(* CoDeSys 2.3.9.55 project: BarCode.pro *)
(* Libraries: STANDARD.LIB 2.6.14 11:37:46, IECSFC.LIB 2.6.14 11:37:46, ANALYZATION.LIB 2.6.14 11:37:46 *)

(* PLC configuration (modules and I/O channels)
PLC63 [Root] node -1, in %IB0 out %QB0 {BName = #NМеню ПЛК63#A0; MinCycleLenght = 1; MaxCycleLenght = 1000}
  Configuration [ID10050] node 0, in %IB0 out %QB0 {BName = #NКонфигурация#A0}
    DInputs [ID10051] node 0, in %IB0.0 out %QB0.0 {BName = #NДискретные Вх.#A0}
      AT %IB0.0.0 [DInput] Битовая маска входов {CPString128 = #NСост.Дискр.Вх.#Fr.Cn#B0120#A3#O#V2#T02; DinLM = #NЛогика Дискр.Вх#Finv.D#B0121#A0#V2#T02#D00#MFF; DinFl = #NПост.Ф.ДребКонт#FTin.F#B0122#A0#U0017#T02#D0A#MFF}
    Outputs [ID10057] node 1, in %IB0.1 out %QB0.1 {BName = #NВУ#A0}
      AT %QD0.1.0 [AnalogOutput0] Выход 1 {CPString128 = #NСост.ВУ1#Fr.oe#I00#B0000#A0#O#C3#T00#M+1.00E+00; AoutPWMP = #NПериод ШИМ ВУ1#Fthpd#I00#B0123#A0#U0017#T01#D03E8#L0002#MFDE8; AoutPWMM = #NМин.имп.ШИМ ВУ1#Ft.L#I00#B0129#A0#U0017#T01#D0032#L0001#M1388; AoutSafeValue = #NБезоп.сост.ВУ1#FO.ALr#I00#B000C#A0#C3#T00#D+0.00E+00#M+1.00E+00}
      AT %QD0.1.1 [AnalogOutput1] Выход 2 {CPString128 = #NСост.ВУ2#Fr.oe#I01#B0002#A0#O#C3#T00#M+1.00E+00; AoutPWMP = #NПериод ШИМ ВУ2#Fthpd#I01#B0124#A0#U0017#T01#D03E8#L0002#MFDE8; AoutPWMM = #NМин.имп.ШИМ ВУ2#Ft.L#I01#B012A#A0#U0017#T01#D0032#L0001#M1388; AoutSafeValue = #NБезоп.сост.ВУ2#FO.ALr#I01#B000E#A0#C3#T00#D+0.00E+00#M+1.00E+00}
      AT %QD0.1.2 [AnalogOutput2] Выход 3 {CPString128 = #NСост.ВУ3#Fr.oe#I02#B0004#A0#O#C3#T00#M+1.00E+00; AoutPWMP = #NПериод ШИМ ВУ3#Fthpd#I02#B0125#A0#U0017#T01#D03E8#L0002#MFDE8; AoutPWMM = #NМин.имп.ШИМ ВУ3#Ft.L#I02#B012B#A0#U0017#T01#D0032#L0001#M1388; AoutSafeValue = #NБезоп.сост.ВУ3#FO.ALr#I02#B0010#A0#C3#T00#D+0.00E+00#M+1.00E+00}
      AT %QD0.1.3 [AnalogOutput3] Выход 4 {CPString128 = #NСост.ВУ4#Fr.oe#I03#B0006#A0#O#C3#T00#M+1.00E+00; AoutPWMP = #NПериод ШИМ ВУ4#Fthpd#I03#B0126#A0#U0017#T01#D03E8#L0002#MFDE8; AoutPWMM = #NМин.имп.ШИМ ВУ4#Ft.L#I03#B012C#A0#U0017#T01#D0032#L0001#M1388; AoutSafeValue = #NБезоп.сост.ВУ4#FO.ALr#I03#B0012#A0#C3#T00#D+0.00E+00#M+1.00E+00}
      AT %QD0.1.4 [AnalogOutput4] Выход 5 {CPString128 = #NСост.ВУ5#Fr.oe#I04#B0008#A0#O#C3#T00#M+1.00E+00; AoutPWMP = #NПериод ШИМ ВУ5#Fthpd#I04#B0127#A0#U0017#T01#D03E8#L0002#MFDE8; AoutPWMM = #NМин.имп.ШИМ ВУ5#Ft.L#I04#B012D#A0#U0017#T01#D0032#L0001#M1388; AoutSafeValue = #NБезоп.сост.ВУ5#FO.ALr#I04#B0014#A0#C3#T00#D+0.00E+00#M+1.00E+00}
      AT %QD0.1.5 [AnalogOutput5] Выход 6 {CPString128 = #NСост.ВУ6#Fr.oe#I05#B000A#A0#O#C3#T00#M+1.00E+00; AoutPWMP = #NПериод ШИМ ВУ6#Fthpd#I05#B0128#A0#U0017#T01#D03E8#L0002#MFDE8; AoutPWMM = #NМин.имп.ШИМ ВУ6#Ft.L#I05#A0#B012E#U0017#T01#D0032#L0001#M1388; AoutSafeValue = #NБезоп.сост.ВУ6#FO.ALr#I05#B0016#A0#C3#T00#D+0.00E+00#M+1.00E+00}
    AInputs [ID10055] node 2, in %IB0.2 out %QB0.2 {BName = #NАналоговые Вх.#A0; Spay = #NКоррекция ХС#Fcj-.c#B012F#A0#U002A#T03#D01}
      AT %ID0.2.0 [AnalogInput0] Аналоговый вход 1 {CPString128 = #NВход 1#Fread#I00#B0018#C2#A3#O#V3#T10; AinType = #NТип датчика 1#Fin-t#I00#B0130#A0#U002F#T04#D01#M15; InFD = #NПост. фильтра 1#Fin.Fd#I00#B0138#A0#U0018#T01#D0005#M0708; InFG = #NПолоса Фильтра1#Fin.FG#I00#B0028#A0#T00#D+1.00E+01#L+0.00E+01#M+9.99E+03}
      AT %ID0.2.1 [AnalogInputTime0] Время измерения 1
      AT %ID0.2.2 [AnalogInput1] Аналоговый вход 2 {CPString128 = #NВход 2#Fread#I01#B001A#C2#A3#O#V3#T10; AinType = #NТип датчика 2#Fin-t#I01#B0131#A0#U002F#T04#D01#M15; InFD = #NПост. фильтра 2#Fin.Fd#I01#B0139#A0#U0018#T01#D0005#M0708; InFG = #NПолоса Фильтра2#Fin.FG#I01#B002A#A0#T00#D+1.00E+01#L+0.00E+01#M+9.99E+03}
      AT %ID0.2.3 [AnalogInputTime1] Время измерения 2
      AT %ID0.2.4 [AnalogInput2] Аналоговый вход 3 {CPString128 = #NВход 3#Fread#I02#B001C#C2#A3#O#V3#T10; AinType = #NТип датчика 3#Fin-t#I02#B0132#A0#U002F#T04#D01#M15; InFD = #NПост. фильтра 3#Fin.Fd#I02#B013A#A0#U0018#T01#D0005#M0708; InFG = #NПолоса Фильтра3#Fin.FG#I02#B002C#A0#T00#D+1.00E+01#L+0.00E+01#M+9.99E+03}
      AT %ID0.2.5 [AnalogInputTime2] Время измерения 3
      AT %ID0.2.6 [AnalogInput3] Аналоговый вход 4 {CPString128 = #NВход 4#Fread#I03#B001E#C2#A3#O#V3#T10; AinType = #NТип датчика 4#Fin-t#I03#B0133#A0#U002F#T04#D01#M15; InFD = #NПост. фильтра 4#Fin.Fd#I03#B013B#A0#U0018#T01#D0005#M0708; InFG = #NПолоса Фильтра4#Fin.FG#I03#A0#B002E#T00#D+1.00E+01#L+0.00E+01#M+9.99E+03}
      AT %ID0.2.7 [AnalogInputTime3] Время измерения 4
      AT %ID0.2.8 [AnalogInput4] Аналоговый вход 5 {CPString128 = #NВход 5#Fread#I04#B0020#C2#A3#O#V3#T10; AinType = #NТип датчика 5#Fin-t#I04#B0134#A0#U002F#T04#D01#M15; InFD = #NПост. фильтра 5#Fin.Fd#I04#B013C#A0#U0018#T01#D0005#M0708; InFG = #NПолоса Фильтра5#Fin.FG#I04#B0030#A0#T00#D+1.00E+01#L+0.00E+01#M+9.99E+03}
      AT %ID0.2.9 [AnalogInputTime4] Время измерения 5
      AT %ID0.2.10 [AnalogInput5] Аналоговый вход 6 {CPString128 = #NВход 6#Fread#I05#B0022#C2#A3#O#V3#T10; AinType = #NТип датчика 6#Fin-t#I05#B0135#A0#U002F#T04#D01#M15; InFD = #NПост. фильтра 6#Fin.Fd#I05#B013D#A0#U0018#T01#D0005#M0708; InFG = #NПолоса Фильтра6#Fin.FG#I05#B0032#A0#T00#D+1.00E+01#L+0.00E+01#M+9.99E+03}
      AT %ID0.2.11 [AnalogInputTime5] Время измерения 6
      AT %ID0.2.12 [AnalogInput6] Аналоговый вход 7 {CPString128 = #NВход 7#Fread#I06#B0024#C2#A3#O#V3#T10; AinType = #NТип датчика 7#Fin-t#I06#B0136#A0#U002F#T04#D01#M15; InFD = #NПост. фильтра 7#Fin.Fd#I06#B013E#A0#U0018#T01#D0005#M0708; InFG = #NПолоса Фильтра7#Fin.FG#I06#B0034#A0#T00#D+1.00E+01#L+0.00E+01#M+9.99E+03}
      AT %ID0.2.13 [AnalogInputTime6] Время измерения 7
      AT %ID0.2.14 [AnalogInput7] Аналоговый вход 8 {CPString128 = #NВход 8#Fread#I07#B0026#C2#A3#O#V3#T10; AinType = #NТип датчика 8#Fin-t#I07#B0137#A0#U002F#T04#D01#M15; InFD = #NПост. фильтра 8#Fin.Fd#I07#B013F#A0#U0018#T01#D0005#M0708; InFG = #NПолоса Фильтра8#Fin.FG#I07#B0036#A0#T00#D+1.00E+01#L+0.00E+01#M+9.99E+03}
      AT %ID0.2.15 [AnalogInputTime7] Время измерения 8
    MR1_Outputs [ID10053] node 3, in %IB0.3 out %QB0.3 {BName = #NВУ МР1#A0}
      AT %QB0.3.0 [DOutput] ВУ МР1 {CPString128 = #NСост.ВУ МР1#Fr.oe.s#B0140#A0#O#V2#T02}
    Additional [ID10059] node 4, in %IB0.4 out %QB0.4 {BName = #NДоп.пар-ры#A0}
      AT %QB0.4.0 [LCDLight] Подсветка {CPString128 = #NЯрк.подсв.ЖКИ#Find.i#B0141#A0#T02#D2D#M32}
      AT %QB0.4.1 [LCDContrast] Контраст {CPString128 = #NКонтраст ЖКИ#Find.C#B0142#A0#T02#D19#L05#M20}
      AT %IB0.4.2 [KBD] Клавиатура {CPString128 = #NСост.клавиатуры#Fkbrd#B0143#A3#O#T02; KBDBeep = #NЗвук кнопок#Fbeep#B0144#A0#U002A#T03#D01}
      AT %QD0.4.3 [RTS] Часы контроллера {RTSPar = #NВремя и дата#FrtC#B0038#A0#O#T05}
    Versions [ID10060] node 5, in %IB0.5 out %QB0.5 {BName = #NВерсииПрошивок#A0}
      AT %QB0.5.0 [DevName] Имя устройства {CPString128 = #NИмя устройства#Fdev#B003A#A3#O#T08}
      AT %IB0.5.1 [HardVer] Прошивка {CPString128 = #NВерсия прошивки#Fver#B0042#A3#O#T08}
      AT %QB0.5.2 [SoftVer] Программа {CPString128 = #NВерсияПрограммы#Fp.ver#B004A#A3#O#T08}
    RS-485 [ID10061] node 6, in %IB0.6 out %QB0.6 {BName = #NНастр.RS-485#A0; RSBPS = #NСкорость#FbPS#B0145#A0#U0046#T04#D00#M09; RSWLen = #NДлина слова#FLen#B0146#A0#U0005#T04#D03#M03; RSPrt = #NЧётность#Fprty#B0147#A0#U009A#T04#D04#M04; RSStp = #NСтоп биты#Fsbit#B0148#A0#U00A1#T04#D00#M02; RSALen = #NДлина адреса#Fa.len#B0149#A0#U0055#T03#D00; RSAdr = #NАдрес прибора#FAddr#B014A#A0#T01#D0010#M07FF; RSDl = #NЗадержка ответа#FRs.dl#B014B#A0#U0017#T02#D05#M32}
  WorkInd [ID10100] node 1, in %IB1 out %QB1 {WIChanelCount = 6}
  SubMenu [ID11000] node 2, in %IB2 out %QB2 {BName = #NВетка#A0}
  SubMenu [ID11000] node 3, in %IB3 out %QB3 {BName = #NВетка#A0}
  SubMenu [ID11000] node 4, in %IB4 out %QB4 {BName = #NВетка#A0}
*)

(* POU PLC_PRG, ST *)
PROGRAM PLC_PRG
VAR
END_VAR

END_PROGRAM

(* POU FB/fbButtleCounter, ST *)
FUNCTION_BLOCK fbButtleCounter
VAR_INPUT
	xDI					: BOOL;
	wMaxNomber		: WORD:= 5;
END_VAR
VAR_OUTPUT
	wCurrentNumber	: WORD;
END_VAR
VAR
	rtDI				: R_TRIG;
END_VAR
rtDI(CLK:= xDI );

IF rtDI.Q THEN
	IF wCurrentNumber < wMaxNomber  THEN
		wCurrentNumber:= wCurrentNumber + 1;
	ELSE
		wCurrentNumber:= 1;
END_IF
END_FUNCTION_BLOCK
